// TIA Portal V19 export
TYPE "LUC_typeStateCommands"
TITLE = LUC_typeStateModeManagerRequest
// Unit State Commands
// stored: Access Published
   STRUCT
      reset : Bool;   // OMAC PackMLV2022 control command Reset
      start : Bool;   // OMAC PackMLV2022 control command Start
      stop : Bool;   // OMAC PackMLV2022 control command Stop
      hold : Bool;   // OMAC PackMLV2022 control command Hold
      unhold : Bool;   // OMAC PackMLV2022 control command Unhold
      suspend : Bool;   // OMAC PackMLV2022 control command Suspend
      unsuspend : Bool;   // OMAC PackMLV2022 control command Unsuspend
      abort : Bool;   // OMAC PackMLV2022 control command Abort
      clear : Bool;   // OMAC PackMLV2022 control command Clear
      complete : Bool;   // OMAC PackMLV2022 control command Complete
      stateComplete : Bool;   // OMAC PackMLV2022 control command State Complete
   END_STRUCT;
END_TYPE
